{attribute 'qualified_only' := ''}
{attribute 'strict' := ''}
TYPE cDeviceHeading :
(
	Empty := 0,
	Puck := 1,
	Tray := 2,
	Carrier := 3,
	Tote := 4,
	Carton := 5,
	Box := 6,
	Buffer := 20,
	VisionStand := 10,
	ExceptionConv := 11,
	Flipper := 30,
	EvalToolType1 := 31,
	EvalToolType2 := 32,
	JustifyNest1 := 101,
	JustifyNest2 := 102,
	Reject := 998,
	Recovery := 999
) DINT;
END_TYPE

(* stored: Version 1.1.0.1, ProductVersion 3.1.4024.6
   DUT cDeviceHeading: Id {1183befd-81bf-4601-9aef-e089e73ce422} *)
